(* IEC 61131-3 sources: com.logicals.lc3.webinar/usRTS_RPMControl_iSOC/src_FB_LIB_SAFE/Convert/SINT, 4 files *)

(* ---- wSINT_TO_DINT.iecst ---- *)
NAMESPACE logicals.web.standard
NAMESPACE convert

/*
 * Function block wrapper for IEC 61131-3 TO_DINT<br>
 * IN =  input value (SINT)<br>
 * OUT = IN (DINT)<br>
 */
FUNCTION_BLOCK wSINT_TO_DINT
	{ vNameAlignment:="center"; altName:="SINT_TO_DINT"; bgColor:="LightPink"; width:=140; hideIONames; }
	VAR_INPUT
		IN : SINT;
	END_VAR
	VAR_OUTPUT
		OUT: DINT;
	END_VAR

	OUT := TO_DINT(IN:=IN, ENO=>ENO);
END_FUNCTION_BLOCK

END_NAMESPACE
END_NAMESPACE

(* ---- wSINT_TO_INT.iecst ---- *)
NAMESPACE logicals.web.standard
NAMESPACE convert

/*
 * Function block wrapper for IEC 61131-3 TO_INT<br>
 * IN =  input value (SINT)<br>
 * OUT = IN (INT)<br>
 */
FUNCTION_BLOCK wSINT_TO_INT
	{ vNameAlignment:="center"; altName:="SINT_TO_INT"; bgColor:="LightPink"; width:=140; hideIONames; }
	VAR_INPUT
		IN : SINT;
	END_VAR
	VAR_OUTPUT
		OUT: INT;
	END_VAR

	OUT := TO_INT(IN:=IN, ENO=>ENO);
END_FUNCTION_BLOCK

END_NAMESPACE
END_NAMESPACE

(* ---- wSINT_TO_LINT.iecst ---- *)
NAMESPACE logicals.web.standard
NAMESPACE convert

/*
 * Function block wrapper for IEC 61131-3 TO_LINT<br>
 * IN =  input value (SINT)<br>
 * OUT = IN (LINT)<br>
 */
FUNCTION_BLOCK wSINT_TO_LINT
	{ vNameAlignment:="center"; altName:="SINT_TO_LINT"; bgColor:="LightPink"; width:=140; hideIONames; }
	VAR_INPUT
		IN : SINT;
	END_VAR
	VAR_OUTPUT
		OUT: LINT;
	END_VAR

	OUT := TO_LINT(IN:=IN, ENO=>ENO);
END_FUNCTION_BLOCK

END_NAMESPACE
END_NAMESPACE

(* ---- wTRUNC_SINT_TO_USINT.iecst ---- *)
NAMESPACE logicals.web.standard
NAMESPACE convert

/*
 * Function block wrapper for IEC 61131-3 TO_USINT<br>
 * IN =  input value (SINT)<br>
 * OUT = IN (USINT)<br>
 */
FUNCTION_BLOCK wTRUNC_SINT_TO_USINT
	{ vNameAlignment:="center"; altName:="TRUNC_SINT_TO_USINT"; bgColor:="Plum"; width:=180; hideIONames; }
	VAR_INPUT
		IN : SINT;
	END_VAR
	VAR_OUTPUT
		OUT: USINT;
	END_VAR

	OUT := TO_USINT(IN:=IN, ENO=>ENO);
END_FUNCTION_BLOCK

END_NAMESPACE
END_NAMESPACE
